//project related global constants
{attribute 'qualified_only'}
VAR_GLOBAL CONSTANT

{info 'TODO: TEMPLATE REMOVE WHEN NOT NEEDED'}
//array sizes >> use this to initialise the array AND then use it in the for loops which run through the arrays etc
	//MaxIndexForMyArray:INT:=10;
	//to be used as:
	//MyArray: array[0..MaxIndexForMyArray] of bool;
	//and then
	//FOR index:=0 to MaxIndexForMyArray by 1 DO ...
END_VAR

(* stored: Version 1.1.0.1
   GVL Glcn: Id {f86596d9-1d4b-49d8-8ab9-4b28fda31ccb} *)
